# B&R Automation Studio project warcabot (part 2)

#### Types.typ
```iecst
TYPE
	CameraCommandType : 	STRUCT
		Enable : BOOL;
		AcquireImage : BOOL;
		SearchAcquisitionSettings : BOOL;
	END_STRUCT;
	BoardCalibrationType : 	STRUCT
		BottomRightY : DINT;
		BottomRightX : DINT;
		BottomLeftY : DINT;
		BottomLeftX : DINT;
		TopRightY : DINT;
		TopRightX : DINT;
		TopLeftY : DINT;
		TopLeftX : DINT;
		MarkersValid : BOOL;
		ReferenceMarker4Y : DINT;
		ReferenceMarker4X : DINT;
		ReferenceMarker3Y : DINT;
		ReferenceMarker3X : DINT;
		ReferenceBottomRightY : DINT;
		ReferenceBottomRightX : DINT;
		ReferenceBottomLeftY : DINT;
		ReferenceBottomLeftX : DINT;
		ReferenceTopRightY : DINT;
		ReferenceTopRightX : DINT;
		ReferenceTopLeftY : DINT;
		ReferenceTopLeftX : DINT;
	END_STRUCT;
	CameraParameterType : 	STRUCT
		FlashColor : USINT;
		FlashSegment : USINT;
		SetFocus : UINT;
		ExposureTime : UDINT;
		NumSearchMax : USINT;
		ScoreMin : USINT;
		GainLevel : USINT;
	END_STRUCT;
	CameraStatusType : 	STRUCT
		AcquisitionReady : BOOL;
		ProcessingActive : BOOL;
		ProcessingError : UINT;
		ReadFocus : UINT;
		ReadExposureTime : UDINT;
		ReadGainLevel : USINT;
	END_STRUCT;
	DetectedPieceType : 	STRUCT
		PositionX : DINT;
		PositionY : DINT;
		Valid : BOOL;
		Score : USINT;
		ModelNumber : USINT;
		Column : USINT;
		Row : USINT;
	END_STRUCT;
	CameraBoardType :ARRAY[1..8,1..8]OF USINT;
	CameraControlType : 	STRUCT
		Cmd : CameraCommandType;
		Parameters : CameraParameterType;
		Status : CameraStatusType;
		NumResults : USINT;
		Pieces : ARRAY[1..26]OF DetectedPieceType;
		Calibration : BoardCalibrationType;
		Board : CameraBoardType;
		BoardReady : BOOL;
		BlackCount : USINT;
		WhiteCount : USINT;
		BoardDataValid : BOOL;
	END_STRUCT;
END_TYPE
```

#### Variables.var
```iecst
VAR
	marker4X : DINT;
	marker3Y : DINT;
	marker3X : DINT;
	j : USINT;
	currentRightX : DINT;
	currentBoardWidth : DINT;
	currentLeftX : DINT;
	boardHeight : DINT;
	PreviousCameraAutoAdjust : BOOL;
	i : USINT;
	gCameraCtrl : CameraControlType;
	PreviousProcessingActive : BOOL;
	columnIndex : USINT;
	rowIndex : USINT;
	cellStepY : DINT;
	cellStepX : DINT;
	relativeY : DINT;
	relativeX : DINT;
	transformedY : LREAL;
	transformedX : LREAL;
	cornerRelativeY : LREAL;
	cornerRelativeX : LREAL;
	transformationDen : LREAL;
	transformationB : LREAL;
	transformationA : LREAL;
	currentVectorY : LREAL;
	currentVectorX : LREAL;
	referenceVectorY : LREAL;
	referenceVectorX : LREAL;
	marker4Found : BOOL;
	marker3Found : BOOL;
	marker4Y : DINT;
	PreviousAutoProcessingActive : BOOL;
END_VAR
```

#### Main.st
```iecst
PROGRAM _INIT

	gCameraCtrl.Cmd.Enable := TRUE;
	gCameraCtrl.Cmd.AcquireImage := FALSE;

	gCameraAutoAdjust := FALSE;
	PreviousCameraAutoAdjust := FALSE;

	gCameraExposureTime := 20884;
	gCameraGainLevel := 4;
	gCameraFocus := 53073;

	gCameraCtrl.Parameters.ExposureTime := gCameraExposureTime;
	gCameraCtrl.Parameters.SetFocus := gCameraFocus;
	gCameraCtrl.Parameters.GainLevel := gCameraGainLevel;
	gCameraCtrl.Parameters.FlashColor := 3;
	gCameraCtrl.Parameters.FlashSegment := 1;

	gCameraCtrl.Parameters.ScoreMin := 75;
	gCameraCtrl.Parameters.NumSearchMax := 26;

	gCameraCtrl.Calibration.ReferenceTopLeftX := 41009;
	gCameraCtrl.Calibration.ReferenceTopLeftY := 14517;
	gCameraCtrl.Calibration.ReferenceTopRightX := 120526;
	gCameraCtrl.Calibration.ReferenceTopRightY := 12412;

	gCameraCtrl.Calibration.ReferenceBottomLeftX := 41915;
	gCameraCtrl.Calibration.ReferenceBottomLeftY := 91572;

	gCameraCtrl.Calibration.ReferenceBottomRightX := 121154;
	gCameraCtrl.Calibration.ReferenceBottomRightY := 90368;

	gCameraCtrl.Calibration.ReferenceMarker3X := 41009;
	gCameraCtrl.Calibration.ReferenceMarker3Y := 14517;

	gCameraCtrl.Calibration.ReferenceMarker4X := 121154;
	gCameraCtrl.Calibration.ReferenceMarker4Y := 90368;

	gCameraCtrl.Calibration.MarkersValid := FALSE;

	gCameraCtrl.BoardReady := FALSE;
	gCameraCtrl.BoardDataValid := FALSE;
	gCameraCtrl.WhiteCount := 0;
	gCameraCtrl.BlackCount := 0;

	gCameraEnd := FALSE;
	PreviousProcessingActive := FALSE;

END_PROGRAM

PROGRAM _CYCLIC

	gCameraCtrl.Cmd.Enable := TRUE;

	(* Wyświetlanie rzeczywistych wartości kamery *)
	gCameraReadExposureTime :=
	gCameraCtrl.Status.ReadExposureTime;

	gCameraReadGainLevel :=
	gCameraCtrl.Status.ReadGainLevel;

	gCameraReadFocus :=
	gCameraCtrl.Status.ReadFocus;

	(* Po wyłączeniu ustawiania zapisz znalezione parametry *)
	IF PreviousCameraAutoAdjust AND NOT gCameraAutoAdjust THEN

		gCameraExposureTime :=
		gCameraCtrl.Status.ReadExposureTime;

		gCameraGainLevel :=
		gCameraCtrl.Status.ReadGainLevel;

		gCameraFocus :=
		gCameraCtrl.Status.ReadFocus;

	END_IF;

	(* Poza automatycznym ustawianiem wysyłaj zapisane nastawy *)
	IF NOT gCameraAutoAdjust THEN

		gCameraCtrl.Parameters.ExposureTime :=
		gCameraExposureTime;

		gCameraCtrl.Parameters.GainLevel :=
		gCameraGainLevel;

		gCameraCtrl.Parameters.SetFocus :=
		gCameraFocus;

	END_IF;

	PreviousCameraAutoAdjust := gCameraAutoAdjust;

	IF gCameraTrigger
		AND NOT gCameraAutoAdjust
		AND NOT gCameraEnd
		AND gCameraCtrl.Status.AcquisitionReady
		AND NOT gCameraCtrl.Status.ProcessingActive
		AND (gCameraCtrl.Status.ProcessingError = 0) THEN
		gCameraCtrl.Cmd.AcquireImage := TRUE;
	END_IF;

	gCameraBlackCount := gCameraCtrl.BlackCount;
	gCameraWhiteCount := gCameraCtrl.WhiteCount;
	gCameraNumResults := gCameraCtrl.NumResults;

	IF NOT gCameraTrigger THEN
		gCameraCtrl.Cmd.AcquireImage := FALSE;
		gCameraCtrl.BoardReady := FALSE;
		gCameraCtrl.BoardDataValid := FALSE;
		gCameraEnd := FALSE;
	END_IF;

	IF gCameraCtrl.Status.ProcessingActive THEN
		gCameraCtrl.Cmd.AcquireImage := FALSE;
	END_IF;

	IF gCameraTrigger
		AND PreviousProcessingActive
		AND NOT gCameraCtrl.Status.ProcessingActive THEN
		gCameraCtrl.Cmd.AcquireImage := FALSE;
		gCameraCtrl.BoardDataValid := TRUE;
		gCameraCtrl.WhiteCount := 0;
		gCameraCtrl.BlackCount := 0;
		marker3Found := FALSE;
		marker4Found := FALSE;
		cellStepY := 0;

		FOR rowIndex := 1 TO 8 DO
			FOR columnIndex := 1 TO 8 DO
				gCameraCtrl.Board[rowIndex, columnIndex] := 0;
			END_FOR;
		END_FOR;

		FOR i := 1 TO 26 DO
			IF gCameraCtrl.NumResults >= i THEN

				IF (gCameraCtrl.Pieces[i].ModelNumber = 3)
					AND (gCameraCtrl.Pieces[i].Score >= 30) THEN

					IF NOT marker3Found THEN

						marker3X := gCameraCtrl.Pieces[i].PositionX;
						marker3Y := gCameraCtrl.Pieces[i].PositionY;

						marker4X := gCameraCtrl.Pieces[i].PositionX;
						marker4Y := gCameraCtrl.Pieces[i].PositionY;

						marker3Found := TRUE;

					ELSE

						IF gCameraCtrl.Pieces[i].PositionX < marker3X THEN

							marker4X := marker3X;
							marker4Y := marker3Y;

							marker3X := gCameraCtrl.Pieces[i].PositionX;
							marker3Y := gCameraCtrl.Pieces[i].PositionY;

						ELSIF gCameraCtrl.Pieces[i].PositionX > marker4X THEN

							marker4X := gCameraCtrl.Pieces[i].PositionX;
							marker4Y := gCameraCtrl.Pieces[i].PositionY;

						END_IF;

						marker4Found := TRUE;

					END_IF;

				END_IF;

			END_IF;
		END_FOR;

		gCameraCtrl.Calibration.MarkersValid := marker3Found AND marker4Found;

		IF gCameraCtrl.Calibration.MarkersValid THEN
			referenceVectorX := DINT_TO_LREAL(gCameraCtrl.Calibration.ReferenceMarker4X- gCameraCtrl.Calibration.ReferenceMarker3X);

			referenceVectorY := DINT_TO_LREAL(gCameraCtrl.Calibration.ReferenceMarker4Y- gCameraCtrl.Calibration.ReferenceMarker3Y);

			currentVectorX := DINT_TO_LREAL(marker4X - marker3X);

			currentVectorY := DINT_TO_LREAL(marker4Y - marker3Y);

			transformationDen := (referenceVectorX * referenceVectorX) + (referenceVectorY * referenceVectorY);

			IF transformationDen > 0.0 THEN

				transformationA := ((currentVectorX * referenceVectorX) + (currentVectorY * referenceVectorY)) / transformationDen;

				transformationB := ((currentVectorY * referenceVectorX) - (currentVectorX * referenceVectorY)) / transformationDen;

				transformationDen := (transformationA * transformationA) + (transformationB * transformationB);

				IF transformationDen > 0.0 THEN

					boardHeight := ((gCameraCtrl.Calibration.ReferenceBottomLeftY - gCameraCtrl.Calibration.ReferenceTopLeftY) +
					(gCameraCtrl.Calibration.ReferenceBottomRightY - gCameraCtrl.Calibration.ReferenceTopRightY)) / 2;

					IF boardHeight > 0 THEN
						cellStepY := boardHeight / 7;
					ELSE
						gCameraCtrl.BoardDataValid := FALSE;
					END_IF;

				ELSE
					gCameraCtrl.BoardDataValid := FALSE;
				END_IF;

			ELSE
				gCameraCtrl.BoardDataValid := FALSE;
			END_IF;

		ELSE
			gCameraCtrl.BoardDataValid := FALSE;
		END_IF;

		FOR i := 1 TO 26 DO

			gCameraCtrl.Pieces[i].Valid :=
			(gCameraCtrl.NumResults >= i)
			AND
			(gCameraCtrl.Pieces[i].Score >= gCameraCtrl.Parameters.ScoreMin)
			AND
			((gCameraCtrl.Pieces[i].ModelNumber = 1)
			OR
			(gCameraCtrl.Pieces[i].ModelNumber = 2));

			IF gCameraCtrl.Pieces[i].Valid
				AND gCameraCtrl.Calibration.MarkersValid
				AND (cellStepY > 0)
				AND (transformationDen > 0.0) THEN

				cornerRelativeX := DINT_TO_LREAL(gCameraCtrl.Pieces[i].PositionX - marker3X);

				cornerRelativeY := DINT_TO_LREAL(gCameraCtrl.Pieces[i].PositionY - marker3Y);

				transformedX := DINT_TO_LREAL(gCameraCtrl.Calibration.ReferenceMarker3X) +
				((transformationA * cornerRelativeX) + (transformationB * cornerRelativeY)) / transformationDen;

				transformedY := DINT_TO_LREAL(gCameraCtrl.Calibration.ReferenceMarker3Y) +
				((-transformationB * cornerRelativeX) + (transformationA * cornerRelativeY)) / transformationDen;

				relativeY := LREAL_TO_DINT(transformedY) - gCameraCtrl.Calibration.ReferenceTopLeftY;

				IF relativeY < -(cellStepY / 2)
					OR relativeY > (boardHeight + (cellStepY / 2)) THEN

					gCameraCtrl.Pieces[i].Valid := FALSE;
					gCameraCtrl.BoardDataValid := FALSE;

				ELSE

					currentLeftX :=
					LREAL_TO_DINT(
						DINT_TO_LREAL(
					gCameraCtrl.Calibration.ReferenceTopLeftX
					)
					+
					(
					DINT_TO_LREAL(
					gCameraCtrl.Calibration.ReferenceBottomLeftX
					- gCameraCtrl.Calibration.ReferenceTopLeftX
					)
					*
					DINT_TO_LREAL(relativeY)
					)
					/
					DINT_TO_LREAL(boardHeight)
					);

					currentRightX :=
					LREAL_TO_DINT(
						DINT_TO_LREAL(
					gCameraCtrl.Calibration.ReferenceTopRightX
					)
					+
					(
					DINT_TO_LREAL(
					gCameraCtrl.Calibration.ReferenceBottomRightX
					- gCameraCtrl.Calibration.ReferenceTopRightX
					)
					*
					DINT_TO_LREAL(relativeY)
					)
					/
					DINT_TO_LREAL(boardHeight)
					);

					currentBoardWidth := currentRightX - currentLeftX;

					IF currentBoardWidth > 0 THEN
						cellStepX := currentBoardWidth / 7;
					ELSE
						cellStepX := 0;
						gCameraCtrl.Pieces[i].Valid := FALSE;
						gCameraCtrl.BoardDataValid := FALSE;
					END_IF;

					IF gCameraCtrl.Pieces[i].Valid
						AND (cellStepX > 0) THEN

						relativeX :=
						LREAL_TO_DINT(transformedX) - currentLeftX;

						IF relativeX < -(cellStepX / 2)
							OR relativeX > (currentBoardWidth + (cellStepX / 2)) THEN

							gCameraCtrl.Pieces[i].Valid := FALSE;
							gCameraCtrl.BoardDataValid := FALSE;

						ELSE

							gCameraCtrl.Pieces[i].Column := DINT_TO_USINT((relativeX + (cellStepX / 2)) / cellStepX) + 1;

							gCameraCtrl.Pieces[i].Row := 9 - (DINT_TO_USINT((relativeY + (cellStepY / 2)) / cellStepY) + 1);

							IF (gCameraCtrl.Pieces[i].Column = 0)
								OR (gCameraCtrl.Pieces[i].Column > 8)
								OR (gCameraCtrl.Pieces[i].Row = 0)
								OR (gCameraCtrl.Pieces[i].Row > 8) THEN

								gCameraCtrl.Pieces[i].Valid := FALSE;
								gCameraCtrl.BoardDataValid := FALSE;

							ELSIF gCameraCtrl.Board[
								gCameraCtrl.Pieces[i].Row,
								gCameraCtrl.Pieces[i].Column
								] <> 0 THEN

								gCameraCtrl.Pieces[i].Valid := FALSE;
								gCameraCtrl.BoardDataValid := FALSE;

							ELSE

								gCameraCtrl.Board[
								gCameraCtrl.Pieces[i].Row,
								gCameraCtrl.Pieces[i].Column
								] :=
								gCameraCtrl.Pieces[i].ModelNumber;

								IF gCameraCtrl.Pieces[i].ModelNumber = 1 THEN
									gCameraCtrl.WhiteCount :=
									gCameraCtrl.WhiteCount + 1;
								ELSE
									gCameraCtrl.BlackCount :=
									gCameraCtrl.BlackCount + 1;
								END_IF;

							END_IF;

						END_IF;

					END_IF;

				END_IF;

			ELSE
				gCameraCtrl.Pieces[i].Valid := FALSE;
			END_IF;

			IF NOT gCameraCtrl.Pieces[i].Valid THEN
				gCameraCtrl.Pieces[i].Row := 0;
				gCameraCtrl.Pieces[i].Column := 0;
			END_IF;

		END_FOR;

		FOR rowIndex := 1 TO 8 DO
			FOR columnIndex := 1 TO 8 DO
				gBoardCamera[rowIndex, columnIndex] :=
				gCameraCtrl.Board[rowIndex, columnIndex];
			END_FOR;
		END_FOR;

		gCameraCtrl.BoardReady :=
		gCameraCtrl.BoardDataValid
		AND (gCameraCtrl.Status.ProcessingError = 0);
		gCameraEnd := TRUE;
	END_IF;

	PreviousProcessingActive := gCameraCtrl.Status.ProcessingActive;

	IF gCameraTrigger
		AND (gCameraCtrl.Status.ProcessingError <> 0) THEN
		gCameraCtrl.Cmd.AcquireImage := FALSE;
		gCameraCtrl.BoardReady := FALSE;
		gCameraCtrl.BoardDataValid := FALSE;
		gCameraEnd := TRUE;
	END_IF;

END_PROGRAM

PROGRAM _EXIT

	gCameraCtrl.Cmd.AcquireImage := FALSE;
	gCameraCtrl.Cmd.Enable := FALSE;

	gCameraCtrl.BoardReady := FALSE;
	gCameraCtrl.BoardDataValid := FALSE;
	gCameraCtrl.Calibration.MarkersValid := FALSE;

	gCameraEnd := FALSE;
	PreviousProcessingActive := FALSE;
	PreviousCameraAutoAdjust := FALSE;
	gCameraAutoAdjust := FALSE;

END_PROGRAM
```

### Program Logical/Programs/SaveGame (IEC)

#### Main.st - Init, cyclic, exit code
```iecst
PROGRAM _INIT
	(* Włączenie Bloków Funkcyjnych MpRecipe *)
	MpRecipeXml_0(MpLink := ADR(MpLinkgRecipeSR), Enable := TRUE, DeviceName := ADR('SG'), FileName := ADR('Save'));
	MpRecipeRegPar_0(MpLink := ADR(MpLinkgRecipeSR), Enable := TRUE, PVName := ADR('SaveGame:Save'));

	(* Włączenie Bloków Funkcyjnych z UI *)
	MpRecipeUI_0(MpLink := ADR(MpLinkgRecipeSR), Enable := TRUE, DeviceName := ADR('SG'), UIConnect := ADR(UIConnect));
	UIConnect.Recipe.SortOrder := mpRECIPE_UI_SORT_DATE_DESCENDING;

END_PROGRAM

PROGRAM _CYCLIC
	(* Function Bloki *)
	MpRecipeXml_0();
	MpRecipeRegPar_0();
	MpRecipeUI_0();

	(* Czyszczenie komunikatów po otwrciu / zamknięciu okna *)
	IF NSDialogOpen THEN
		Saved := FALSE;
		InvSavFileName := FALSE;
		NSDialogOpen := FALSE;
	END_IF;

	CurrentFileName := UIConnect.Recipe.List.Names[UIConnect.Recipe.List.SelectedIndex];

	(* Sprawdzanie czy jest mniej plików niż max *)
	IndexOOR := UIConnect.Recipe.List.MaxSelection >= 19;
	NIndexOOR := UIConnect.Recipe.List.MaxSelection < 19;

	(* Zabezpieczenie przed ingerencją w Function Blok podczas jego pracy *)
	IF UIConnect.Status = mpRECIPE_UI_STATUS_IDLE THEN

		(* Jeśli przycisk New save kliknięty i jest mniej niż max plików
		sprawdź nazwę i możliwie stwórz nowy plik. Wyświetl komunikaty *)
		IF NewSave AND NOT IndexOOR THEN
			Saved := FALSE;
			InvSavFileName := FALSE;
			FB_ValidateFileName_0(sUserInput := SaveFileName);
			IF FB_ValidateFileName_0.bIsValid THEN
				Save.BoardActual := gBoardActual;
				Save.PlayerColor := gPlayerColor;
				Save.DifficultyLevel := gDifficultyLevel;
				Save.MoveHistory := gGameStats.MoveHistory;
				Save.MoveCount := gGameStats.MoveCount;

				UIConnect.New.FileName := FB_ValidateFileName_0.sValidName;
				UIConnect.New.Create := TRUE;
				SaveFileName := '';
				Saved := TRUE;
				NewSave := FALSE;
			ELSE
				InvSavFileName := TRUE;
				NewSave := FALSE;
			END_IF;

		END_IF;

		(* Ładowanie do zmiennej *)
		IF PreLoad THEN
			UIConnect.Recipe.Load := TRUE;
			PreLoad := FALSE;
		END_IF;

		(* Jeśli przycisk Load kliknięty przypisz zmienną z danymi do zmiennej globalnej *)
		IF Load THEN
			gBoardActual := Save.BoardActual;
			gPlayerColor := Save.PlayerColor;
			gDifficultyLevel := Save.DifficultyLevel;
			gGameStats.MoveHistory := Save.MoveHistory;
			gGameStats.MoveCount := Save.MoveCount;

			LoadingDone := TRUE;
			gStart := TRUE;
			gGameStats.Load := TRUE;
			Load := FALSE;
		END_IF;

		(* Jeśli przycisk Delete kliknięty usuń plik o wybranym indeksie *)
		IF DeleteSave THEN
			UIConnect.Recipe.Delete := TRUE;
			DeleteSave := FALSE;
		END_IF
	END_IF;

END_PROGRAM

PROGRAM _EXIT
	(* Wyłączenie Function Bloków *)
	MpRecipeXml_0(Enable := FALSE);
	MpRecipeRegPar_0(Enable := FALSE);
	MpRecipeUI_0(Enable := FALSE);

END_PROGRAM
```

#### Types.typ - Local data types
```iecst
TYPE
	Save_type : 	STRUCT
		BoardActual : ARRAY[1..8,1..8]OF USINT := [2,0,2,0,2,0,2,2(0),2,0,2,0,2,0,2(2),0,2,0,2,0,2,18(0),1,0,1,0,1,0,2(1),0,1,0,1,0,1,2(0),1,0,1,0,1,0,1];
		PlayerColor : BOOL := FALSE;
		MoveHistory : ARRAY[1..4]OF STRING[20];
		MoveCount : INT;
		DifficultyLevel : USINT := 0;
	END_STRUCT;
END_TYPE
```

#### Variables.var - Local variables
```iecst
VAR
	Load : BOOL := FALSE; (*Zmienna czy przycisk Save został kliknięty*)
	DeleteSave : BOOL := FALSE; (*Zmienna czy przycisk Delete został kliknięty*)
	MpRecipeXml_0 : MpRecipeXml;
	MpRecipeRegPar_0 : MpRecipeRegPar;
	MpRecipeUI_0 : MpRecipeUI; (*MpRecipeUI for UI Connection to the ice cream machine*)
	UIConnect : MpRecipeUIConnectType; (*UI Connection - interfejs do mprecipe*)
	Save : Save_type; (*Zmienna do której są zapisywane i z której są odczytywane dane*)
	SaveFileName : STRING[80]; (*Zmienna do przechowywania wpisanej nazwy pliku*)
	NewSave : BOOL := FALSE; (*Zmienna czy przycisk New save został kliknięty*)
	FB_ValidateFileName_0 : FB_ValidateFileName; (*Function Blok do sprawdzania czy nazwa pliku jest poprawna*)
	InvSavFileName : BOOL := FALSE; (*Zmienna do komunukacji o niepoprawnej nazwie*)
	Saved : BOOL := FALSE; (*Zmienna do komunikacji o pomyślnym zapisaniu pliku*)
	NSDialogOpen : BOOL := FALSE; (*Marker o otworzeniu okna New Save*)
	CurrentFileName : STRING[80]; (*Nazwa aktualnie wybranego pliku*)
	IndexOOR : BOOL; (*Marker o zapełnieniu listy (max 20 plików)*)
	NIndexOOR : BOOL; (*Negacja Markera IndexOOR*)
	LoadingDone : BOOL; (*Marker dla silnika gry*)
	PreLoad : BOOL; (*Zmienna czy przycisk Load (preLoead) został kliknięty*)
END_VAR
```

#### LocalFunctions.fun
```iecst
{REDUND_ERROR} FUNCTION_BLOCK FB_ValidateFileName (*Validating file name*) (*$GROUP=User,$CAT=User,$GROUPICON=User.png,$CATICON=User.png*)
	VAR_INPUT
		sUserInput : {REDUND_UNREPLICABLE} STRING[80]; (*Zmienna wejściowa ze sprawdzaną nazwą pliku*)
	END_VAR
	VAR_OUTPUT
		sValidName : STRING[80]; (*Zmienna wyjściowa z poprawną nazwą pliku*)
		bIsValid : BOOL; (*Zmienna informująca czy była możliwość dana poprawnej nazwy pliku na wyjściu*)
	END_VAR
	VAR
		i : UDINT; (*zmienna do iteracji po stringu*)
		tempChar : BYTE; (*Zmienna do przechowywania akutalnie iterownaje litery*)
	END_VAR
	VAR CONSTANT
		UNDERSCORE : BYTE := 95; (*ASCII value for '_'*)
	END_VAR
END_FUNCTION_BLOCK
```

#### FB_ValidateFileName.st
```iecst
(* TODO: Add your comment here *)
FUNCTION_BLOCK FB_ValidateFileName
(* Logic *)
	bIsValid := TRUE;
	sValidName := sUserInput;

	// 1. Check for empty input
	IF sUserInput = '' THEN
		bIsValid := FALSE;
	ELSE
		// 2. Sanitize string
		// We use LEN(sValidName) to get the current length of the string
		FOR i := 0 TO brsstrlen(ADR(sValidName)) - 1 DO
			// 1. READ: Copy current character from string into tempChar
			brsmemcpy(ADR(tempChar), ADR(sValidName) + i, 1);

			// 2. CHECK: Use tempChar for all comparisons
			IF tempChar = 32 THEN
				// WRITE: Copy underscore back into the string at position i
				brsmemcpy(ADR(sValidName) + i, ADR(UNDERSCORE), 1);

			ELSIF tempChar = 92 OR tempChar = 47 OR // \ and /
				tempChar = 58 OR tempChar = 42 OR // : and *
				tempChar = 63 OR tempChar = 34 OR // ? and "
				tempChar = 60 OR tempChar = 62 OR // < and >
				tempChar = 124 THEN               // |

				bIsValid := FALSE;
				EXIT;
			END_IF
		END_FOR
	END_IF
END_FUNCTION_BLOCK
```

### Program Logical/Programs/AlarmHistory (IEC)

#### Variables.var
```iecst
VAR
	AlarmTest : INT := 0; (*Testowa zmienna do testowania alarmów*)
	MpAlarmXHistory_0 : MpAlarmXHistory; (*Function blok MpAlarmXHistory*)
	AHExport : BOOL := FALSE; (*Zmienna czy przycisk export został kliknięty*)
	DirCreate_0 : DirCreate; (*Function Blok tworzący folder*)
	OpenExportDialog : BOOL := FALSE; (*Zmienna, która otwiera okienko z inf o exporcie*)
	AHClear : BOOL;
END_VAR
```

#### Main.st
```iecst
PROGRAM _INIT
	(* Włączenie Function Bloku MpAlarmXHistory *)
	MpAlarmXHistory_0(MpLink := ADR(MpLinkgAlarmXHistory), Enable := TRUE, DeviceName := ADR('AH'), FileName := ADR('Alarm_history'));

END_PROGRAM

PROGRAM _CYCLIC
	MpAlarmXHistory_0();

	(* Jeśli MpAlarmXHistory nic nie robi, a przycisk export kliknięty -> wyexportuj i otwórz okno dialogowe *)
	IF AHExport AND NOT MpAlarmXHistory_0.CommandBusy THEN
		MpAlarmXHistory_0.Export := TRUE;
		IF MpAlarmXHistory_0.CommandDone THEN
			MpAlarmXHistory_0.Export := FALSE;
			OpenExportDialog := TRUE;
			AHExport := FALSE;
		END_IF;
	END_IF;

	IF AHClear AND NOT MpAlarmXHistory_0.CommandBusy THEN
		MpAlarmXHistory_0.Clear := TRUE;
		IF MpAlarmXHistory_0.CommandDone THEN
			AHClear := FALSE;
		END_IF;
	END_IF;

END_PROGRAM

PROGRAM _EXIT
	(* Wyłacz MpAlarmXHistory *)
	MpAlarmXHistory_0(Enable := FALSE);

END_PROGRAM
```

### Program Logical/Programs/VisVariable (IEC)

#### Main.st
```iecst
PROGRAM _INIT
	gPickPiece;
	gEnableMove;
	gPickMove;
	gBoardActual;
	gGameRound;
	gEnablePiece;

END_PROGRAM

PROGRAM _CYCLIC
	(* Insert code here *)

END_PROGRAM

PROGRAM _EXIT
	(* Insert code here *)

END_PROGRAM
```

### Program Logical/Programs/GameStats (IEC)

#### Variables.var
```iecst
VAR
	WinOrLose : BOOL; (*True - wygrana, False - przegrana*)
	EndGame : BOOL; (*True - Koniec gry, False - gra wciaz trwa*)
	DeadWhitePiece : INT; (*Zbite biale pionki*)
	DeadBlackPiece : INT; (*Zbite czarne pionki*)
	MoveCount : INT; (*Ilosc ruchow*)
	i : USINT; (*zmienna do for*)
	j : USINT; (*zmienna do for*)
	whiteOnBoard : INT; (*ilosc bialych pionkow na planszy*)
	blackOnBoard : INT; (*ilosc czarnych pionkow na planszy*)
	gBoardLast : ARRAY[1..8,1..8] OF USINT; (*poprzedni stan planszy*)
	firstScan : BOOL := TRUE; (*pierwszy cykl - tylko zapamietaj plansze*)
	fromRow : USINT; (*wiersz startowy ruchu*)
	fromCol : USINT; (*kolumna startowa ruchu*)
	toRow : USINT; (*wiersz docelowy ruchu*)
	toCol : USINT; (*kolumna docelowa ruchu*)
	capCount : USINT; (*ilosc zbic w ruchu*)
	movedColor : USINT; (*1 - bialy, 2 - czarny*)
	cellColor : USINT; (*kolor pionka na polu*)
	pChar : REFERENCE TO USINT; (*wskaznik do budowy stringu*)
	LastMove : STRING[20]; (*ostatni wykryty ruch*)
	MoveHistory : ARRAY[1..4] OF STRING[20]; (*[1] najnowszy, [4] najstarszy*)
	MpAuditTrail_0 : MpAuditTrail;
	auditTmp : STRING[80];
	MessageVar : WSTRING[100];
	TypeVar : WSTRING[100];
	CommentVar : WSTRING[100];
	MpReportCore_0 : MpReportCore;
	sReport_Color     : STRING[20];
	sReport_Difficulty: STRING[30];
	sReport_Result    : STRING[20];
END_VAR
```

#### Main.st
```iecst
PROGRAM _INIT

	WinOrLose;
	EndGame;
	gPlayerColor;
	gDifficultyLevel;
	gStart;
	gBoardActual;
	j;
	i;
	whiteOnBoard;
	blackOnBoard;
	gEnablePiece;
	sReport_Color;
	sReport_Difficulty;
	sReport_Result;

	gBoardLast := gBoardActual;
	firstScan := TRUE;
	MoveHistory[1] := '';
	MoveHistory[2] := '';
	MoveHistory[3] := '';
	MoveHistory[4] := '';
	LastMove := '';
	MoveCount := 0;

	MpReportCore_0();
	MpReportCore_0.Enable := TRUE;
	MpReportCore_0.MpLink := ADR(gReport);
	MpReportCore_0.DeviceName := ADR('CF');
	MpReportCore_0.FileName := ADR('GameReport');
	MpReportCore_0.ReportID := ADR('MyReport');
	MpReportCore_0.Language := ADR('en');

END_PROGRAM

PROGRAM _CYCLIC

	MpReportCore_0();

	(* --- MAPOWANIE DANYCH NA TEKSTY --- *)

	(* Kolor *)
	IF gPlayerColor THEN
		sReport_Color := 'White';
	ELSE
		sReport_Color := 'Black';
	END_IF;

	(* Poziom trudności *)
	CASE gDifficultyLevel OF
		4: sReport_Difficulty := 'No stress';
		3: sReport_Difficulty := 'Easy going';
		0: sReport_Difficulty := 'Challenge';
		1: sReport_Difficulty := 'Blood, sweat & tears';
		2: sReport_Difficulty := 'Good luck ...';
		ELSE
			sReport_Difficulty := 'Unknown';
	END_CASE;

	(* Wynik *)
	IF WinOrLose THEN
		sReport_Result := 'Victory';
	ELSE
		sReport_Result := 'Defeat';
	END_IF;

	(* --- STEROWANIE GENEROWANIEM RAPORTU --- *)
	IF EndGame AND NOT MpReportCore_0.CommandBusy THEN
		MpReportCore_0.Generate := TRUE;
	ELSE
		MpReportCore_0.Generate := FALSE;
	END_IF;

	IF gStart THEN
		IF gGameStats.Load THEN
			MoveHistory := gGameStats.MoveHistory;
			MoveCount := gGameStats.MoveCount;
			gGameStats.Load := FALSE;
		END_IF;

		whiteOnBoard := 0;
		blackOnBoard := 0;

		FOR i := 1 TO 8 DO
			FOR j := 1 TO 8 DO
				CASE gBoardActual[i, j] OF
					1, 3:  whiteOnBoard := whiteOnBoard + 1;
					2, 4:  blackOnBoard := blackOnBoard + 1;
				END_CASE;
			END_FOR;
		END_FOR;

		DeadWhitePiece := 12 - whiteOnBoard;
		DeadBlackPiece := 12 - blackOnBoard;

		IF firstScan THEN
			gBoardLast := gBoardActual;
			firstScan := FALSE;
		ELSE
			fromRow := 0; fromCol := 0;
			toRow := 0;   toCol := 0;
			capCount := 0;
			movedColor := 0;

			FOR i := 1 TO 8 DO
				FOR j := 1 TO 8 DO
					IF gBoardLast[i, j] = 0 AND gBoardActual[i, j] <> 0 THEN
						toRow := i;
						toCol := j;
						IF gBoardActual[i, j] = 1 OR gBoardActual[i, j] = 3 THEN
							movedColor := 1;
						ELSE
							movedColor := 2;
						END_IF;
					END_IF;
				END_FOR;
			END_FOR;

			IF toRow <> 0 THEN
				FOR i := 1 TO 8 DO
					FOR j := 1 TO 8 DO
						IF gBoardLast[i, j] <> 0 AND gBoardActual[i, j] = 0 THEN
							IF gBoardLast[i, j] = 1 OR gBoardLast[i, j] = 3 THEN
								cellColor := 1;
							ELSE
								cellColor := 2;
							END_IF;

							IF cellColor = movedColor THEN
								fromRow := i;
								fromCol := j;
							ELSE
								capCount := capCount + 1;
							END_IF;
						END_IF;
					END_FOR;
				END_FOR;
			END_IF;

			IF toRow <> 0 AND fromRow <> 0 THEN

				gRobotMoveVar.StartPoint.x := fromCol;
				gRobotMoveVar.StartPoint.y := fromRow;
				gRobotMoveVar.EndPoint.x := toCol;
				gRobotMoveVar.EndPoint.y := toRow;
				gRobotMoveVar.RTRMove := TRUE;

				pChar ACCESS ADR(LastMove);
				pChar := 64 + fromCol;

				pChar ACCESS ADR(LastMove) + 1;
				pChar := 48 + fromRow;

				pChar ACCESS ADR(LastMove) + 2;
				IF capCount > 0 THEN
					pChar := 120;
					gRobotMoveVar.Capture := TRUE;
					gRobotMoveVar.DiscardPoint.x := (fromCol+toCol)/2;
					gRobotMoveVar.DiscardPoint.y := (fromRow+toRow)/2;
					gRobotMoveVar.DiscardColor := (movedColor) MOD 2 + 1;
				ELSE
					pChar := 45;
					gRobotMoveVar.Capture := FALSE;
				END_IF;

				pChar ACCESS ADR(LastMove) + 3;
				pChar := 64 + toCol;

				pChar ACCESS ADR(LastMove) + 4;
				pChar := 48 + toRow;

				pChar ACCESS ADR(LastMove) + 5;
				pChar := 0;

				MoveHistory[4] := MoveHistory[3];
				MoveHistory[3] := MoveHistory[2];
				MoveHistory[2] := MoveHistory[1];
				MoveHistory[1] := LastMove;

				MoveCount := MoveCount + 1;

				(* --- AUDIT: kto wykonal ruch i dokad --- *)
				IF movedColor = gPlayerColor THEN
					brsstrcpy(ADR(auditTmp), ADR('Gracz wykonal ruch: '));
				ELSE
					brsstrcpy(ADR(auditTmp), ADR('Robot wykonal ruch: '));
				END_IF;
				brsstrcat(ADR(auditTmp), ADR(LastMove));

				MessageVar := STRING_TO_WSTRING(auditTmp);
				TypeVar    := "GameMove";
				CommentVar := "";

				MpAuditCustomEvent(gAuditTrail, TypeVar, MessageVar, CommentVar);
				(* --- koniec AUDIT --- *)

				gGameStats.MoveHistory := MoveHistory;
				gGameStats.MoveCount := MoveCount;
			END_IF;

			gBoardLast := gBoardActual;
		END_IF;

	ELSE
		DeadWhitePiece := 0;
		DeadBlackPiece := 0;
		whiteOnBoard := 0;
		blackOnBoard := 0;
		MoveCount := 0;
		LastMove := '';
		MoveHistory[1] := '';
		MoveHistory[2] := '';
		MoveHistory[3] := '';
		MoveHistory[4] := '';
		firstScan := TRUE;
		gBoardLast := gBoardActual;
	END_IF

END_PROGRAM

PROGRAM _EXIT
    (* Insert code here *)

END_PROGRAM
```

### Program Logical/Programs/CheckVision (IEC)

#### Types.typ
```iecst
TYPE
	VisionEnum : 	STRUCT
		BoardConverted : ARRAY[1..8,1..8]OF USINT; (*Przekonwertowana tablica gdzie pokazywany jest tylko kolor, 1 - bialy, 2 - czarny, 0 -brak*)
		BoardVision : ARRAY[1..8,1..8]OF USINT; (*Tablica z kamery *)
		Step : StepVisionEnum; (*Kroki do case*)
		PhotoTake : BOOL; (*TRUE - kamera wykonala zdjecie*)
	END_STRUCT;
	StepVisionEnum :
		(
		CheckTable,
		ConvertTable
		);
END_TYPE
```

#### Variables.var
```iecst
VAR
	OUT : BOOL;
	j : USINT;
	i : USINT;
	Vision : VisionEnum;
	Match : BOOL;
END_VAR
```

#### Main.st
```iecst
PROGRAM _INIT
	gBoardActual;
	Vision;
	OUT := FALSE;

	Match;
	i;
	j;

	Vision.Step := ConvertTable;
	Vision.PhotoTake := FALSE;
END_PROGRAM

PROGRAM _CYCLIC

	CASE Vision.Step OF

		ConvertTable:
			FOR i := 1 TO 8 DO
				FOR j := 1 TO 8 DO
					CASE gBoardActual[i, j] OF
						1:  Vision.BoardConverted[i, j] := 1;
						2:  Vision.BoardConverted[i, j] := 2;
						3:  Vision.BoardConverted[i, j] := 1;
						4:  Vision.BoardConverted[i, j] := 2;
					END_CASE;
				END_FOR;
			END_FOR;

			IF Vision.PhotoTake THEN
				Vision.Step := CheckTable;
			END_IF;

		CheckTable:
			Match := TRUE;
			FOR i := 1 TO 8 DO
				FOR j := 1 TO 8 DO
					IF Vision.BoardConverted[i, j] <> Vision.BoardVision[i, j] THEN
						Match := FALSE;
					END_IF;
				END_FOR;
			END_FOR;

			IF Match THEN
				OUT := TRUE;
				Vision.Step := ConvertTable;
			ELSE
				Vision.Step := ConvertTable;
			END_IF;

	END_CASE

END_PROGRAM

PROGRAM _EXIT
	(* Insert code here *)

END_PROGRAM
```

### Program Logical/Programs/MainProgram (IEC)

#### Types.typ
```iecst
TYPE
	RobotMoveEnum :
		(
		IdleRM,
		MoveExecute,
		MoveBusy,
		DiscardExecute,
		DiscardBusy,
		HomeExecute,
		HomeBusy,
		EndRM
		);
	SetBoardInfoType : 	STRUCT
		Index : IndexPointType;
		Color : USINT; (*White = 1; Black = 2*)
	END_STRUCT;
	SetBoardEnum :
		(
		SetBoardCommandGen,
		SetBoardExecute,
		SetBoardBusy,
		SetBoardHomeExecute,
		SetBoardHomeBusy
		);
	CommandType : 	STRUCT
		EndPos : McPosType;
		StartPos : McPosType;
		EndIndex : IndexPointType;
		StartIndex : IndexPointType;
	END_STRUCT;
END_TYPE
```

#### Variables.var
```iecst
VAR
	ColorCount : ARRAY[1..2] OF USINT := [2(0)];
	MpAuditTrail_0 : MpAuditTrail;
	BoardGit : BOOL; (*Git ruch*)
	Match : BOOL;
	j : USINT;
	i : USINT;
	k : USINT;
	MoveStep : RobotMoveEnum := Idle;
	RobotMoveMarker : BOOL;
	MpReportCore_0 : MpReportCore;
	BuforLastPieceIndex : ARRAY[1..2] OF USINT;
	PiecesToDiscard : ARRAY[1..24] OF SetBoardInfoType;
	DiscardCount : USINT := 0;
	PiecesToDraw : ARRAY[1..24] OF SetBoardInfoType;
	DrawCount : USINT := 0;
	SimBoardValue : USINT := 0;
	CameraBoardValue : USINT := 0;
	DrawHandled : ARRAY[1..24] OF BOOL;
	DiscardHandled : ARRAY[1..24] OF BOOL;
	MatchFound : BOOL := FALSE;
	SetBoardStep : SetBoardEnum := SetBoardCommandGen;
	SetBoardTrigger : BOOL := FALSE;
	RRPCancel : BOOL := FALSE; (*Robot Reset Pos Cancel*)
	RRPConfirm : BOOL := FALSE; (*Robot Reset Pos Confirm*)
	CommandCount : USINT := 0;
	CommandList : ARRAY[1..48] OF CommandType;
	CommandDoneCount : USINT := 0;
	ReportLanguage : STRING[20] := 'en';
	RRPTrigger : BOOL;
END_VAR
VAR CONSTANT
	BOARD_SPACES : USINT := 8;
	CONVERT_BOARD : ARRAY[0..4] OF USINT := [0,1,2,1,2];
	BUFOR_POSITION : ARRAY[1..2,1..12] OF McPosType := [
	(X:=-61.8, Y:=68.9, Z:=-0.5),
	(X:=-28.1, Y:=69.0, Z:=-0.5),
	(X:=4.8, Y:=68.9, Z:=-0.5),
	(X:=-61.4, Y:=105.2, Z:=-0.7),
	(X:=-27.6, Y:=105.4, Z:=-0.8),
	(X:=4.3, Y:=105.2, Z:=-0.7),
	(X:=-61.5, Y:=141.4, Z:=-0.8),
	(X:=-28.4, Y:=141.5, Z:=-0.8),
	(X:=3.4, Y:=141.4, Z:=-0.8),
	(X:=-61.9, Y:=177.5, Z:=-0.9),
	(X:=-29.5, Y:=177.6, Z:=-0.9),
	(X:=2.2, Y:=177.5, Z:=-0.9),
	(X:=426.3, Y:=66.3, Z:=1.9),
	(X:=459.6, Y:=66.3, Z:=1.8),
	(X:=492.9, Y:=66.4, Z:=1.9),
	(X:=426.5, Y:=102.8, Z:=1.7),
	(X:=459.6, Y:=102.8, Z:=1.5),
	(X:=492.7, Y:=102.9, Z:=1.7),
	(X:=426.7, Y:=139.4, Z:=1.6),
	(X:=459.6, Y:=139.5, Z:=1.5),
	(X:=492.4, Y:=139.4, Z:=1.6),
	(X:=426.8, Y:=175.9, Z:=1.5),
	(X:=459.5, Y:=175.9, Z:=1.4),
	(X:=492.1, Y:=175.9, Z:=1.5)
	];
	COORD_POSITION : ARRAY[1..8,1..8] OF McPosType := [
	(X:=62.9, Y:=-29.7, Z:=2.4),
	(X:=107.2, Y:=-26.3, Z:=2.3),
	(X:=150.1, Y:=-26.9, Z:=2.5),
	(X:=193.0, Y:=-27.5, Z:=2.7),
	(X:=236.4, Y:=-28.7, Z:=2.4),
	(X:=278.7, Y:=-28.8, Z:=3.2),
	(X:=321.6, Y:=-29.4, Z:=3.4),
	(X:=363.6, Y:=-28.7, Z:=4.0),
	(X:=64.6, Y:=16.7, Z:=2.5),
	(X:=107.4, Y:=16.1, Z:=2.7),
	(X:=150.3, Y:=15.5, Z:=2.9),
	(X:=193.1, Y:=14.9, Z:=3.1),
	(X:=236.0, Y:=14.3, Z:=3.3),
	(X:=278.8, Y:=13.6, Z:=3.5),
	(X:=321.6, Y:=13.0, Z:=3.7),
	(X:=364.5, Y:=12.4, Z:=3.9),
	(X:=64.8, Y:=59.1, Z:=2.9),
	(X:=107.6, Y:=58.5, Z:=3.1),
	(X:=150.4, Y:=57.9, Z:=3.3),
	(X:=193.2, Y:=57.3, Z:=3.5),
	(X:=236.0, Y:=56.6, Z:=3.7),
	(X:=278.8, Y:=56.0, Z:=3.9),
	(X:=321.6, Y:=55.4, Z:=4.1),
	(X:=364.4, Y:=54.8, Z:=4.3),
	(X:=65.2, Y:=110.4, Z:=3.0),
	(X:=107.9, Y:=100.8, Z:=3.4),
	(X:=150.6, Y:=100.2, Z:=3.6),
	(X:=195.2, Y:=98.9, Z:=3.8),
	(X:=237.6, Y:=98.9, Z:=4.0),
	(X:=278.9, Y:=98.4, Z:=4.3),
	(X:=321.7, Y:=97.8, Z:=4.5),
	(X:=364.4, Y:=97.2, Z:=4.7),
	(X:=65.3, Y:=143.8, Z:=3.6),
	(X:=108.1, Y:=143.2, Z:=3.8),
	(X:=150.8, Y:=142.6, Z:=4.0),
	(X:=193.8, Y:=140.5, Z:=4.6),
	(X:=236.9, Y:=140.5, Z:=4.5),
	(X:=278.9, Y:=140.8, Z:=4.7),
	(X:=321.7, Y:=140.2, Z:=4.9),
	(X:=363.1, Y:=139.0, Z:=4.7),
	(X:=65.6, Y:=186.2, Z:=4.0),
	(X:=108.3, Y:=185.6, Z:=4.2),
	(X:=151.0, Y:=185.0, Z:=4.4),
	(X:=193.6, Y:=184.4, Z:=4.6),
	(X:=236.3, Y:=183.8, Z:=4.8),
	(X:=279.0, Y:=183.2, Z:=5.0),
	(X:=321.7, Y:=182.6, Z:=5.2),
	(X:=364.4, Y:=182.0, Z:=5.4),
	(X:=65.8, Y:=228.5, Z:=4.4),
	(X:=108.5, Y:=227.9, Z:=4.6),
	(X:=151.1, Y:=227.4, Z:=4.8),
	(X:=193.8, Y:=226.8, Z:=5.0),
	(X:=236.4, Y:=226.2, Z:=5.2),
	(X:=279.0, Y:=225.6, Z:=5.4),
	(X:=321.7, Y:=225.0, Z:=5.6),
	(X:=364.3, Y:=224.5, Z:=5.8),
	(X:=65.4, Y:=268.4, Z:=4.7),
	(X:=108.7, Y:=270.3, Z:=4.9),
	(X:=151.3, Y:=269.7, Z:=5.1),
	(X:=193.3, Y:=268.4, Z:=5.4),
	(X:=236.5, Y:=268.6, Z:=5.6),
	(X:=279.1, Y:=268.0, Z:=5.8),
	(X:=321.7, Y:=267.4, Z:=6.0),
	(X:=364.3, Y:=268.4, Z:=6.3)
	];
	DEFAULT_POSITION : McPosType := (X:=-139,Y:=359,Z:=350);
END_VAR
```

#### Main.st
```iecst
PROGRAM _INIT
	gStep := Idle;
	BoardGit := FALSE;

	MpAuditTrail_0.Enable := TRUE;
	MpAuditTrail_0.MpLink := ADR(gAuditTrail);
	MpAuditTrail_0.DeviceName := ADR('AUDIT');
	MpAuditTrail_0.FileName := ADR('AuditList');
	MpAuditTrail_0();
END_PROGRAM

PROGRAM _CYCLIC
	MpAuditTrail_0();

	gStop := NOT gStart;

	IF gESTOP = FALSE THEN
		gMotionInterface.Enable := FALSE;
	END_IF;

	IF gStart = FALSE THEN
		gStep := Idle;
		gRobotMoveVar.RTRMove := FALSE;
		MoveStep := IdleRM;
	END_IF;

	CASE gStep OF
		Idle:
			IF gStart THEN
				SetBoardTrigger := TRUE;
				gStep := ResetRobotPos;
				SetBoardStep := SetBoardBusy;
				gMotionInterface.Enable := TRUE;
				gMotionInterface.RequestManualMode := FALSE;
			END_IF;

		PhotoCheck:
			gCameraTrigger := TRUE;
			IF gCameraEnd THEN
				gCameraTrigger := FALSE;
				Match := TRUE;
				DrawCount := 0;
				DiscardCount := 0;
				ColorCount[1] := 0;
				ColorCount[2] := 0;

				FOR i := 1 TO BOARD_SPACES DO
					FOR j := 1 TO BOARD_SPACES DO
						(* Odwrócenie planszy do góry nogami, aby odczyt z kamery był zgodny z widokiem ze stania na wprost robota *)
						SimBoardValue := CONVERT_BOARD[gBoardActual[i, j]];
						CameraBoardValue := gBoardCamera[BOARD_SPACES + 1 - i, BOARD_SPACES + 1 - j];

						ColorCount[CameraBoardValue] := ColorCount[CameraBoardValue] + 1;

						IF SimBoardValue <> CameraBoardValue THEN
							Match := FALSE;

							IF SetBoardTrigger THEN
								IF CameraBoardValue = 0 THEN
									(* Inkrementujemy najpierw, aby zacząć od indeksu 1 *)
									DrawCount := DrawCount + 1;
									PiecesToDraw[DrawCount].Index.x := i;
									PiecesToDraw[DrawCount].Index.y := j;
									PiecesToDraw[DrawCount].Color := SimBoardValue;
								ELSIF SimBoardValue = 0 THEN
									(* Inkrementujemy najpierw, aby zacząć od indeksu 1 *)
									DiscardCount := DiscardCount + 1;
									PiecesToDiscard[DiscardCount].Index.x := i;
									PiecesToDiscard[DiscardCount].Index.y := j;
									PiecesToDiscard[DiscardCount].Color := CameraBoardValue;
								ELSE
									(* Zarówno w symulacji, jak i w kamerze jest pionek, ale RÓŻNYCH KOLORÓW -> ZAMIANA! *)
									(* 1. Najpierw usuwamy to, co fizycznie stoi na planszy (widzi to kamera) *)
									DiscardCount := DiscardCount + 1;
									PiecesToDiscard[DiscardCount].Index.x := i;
									PiecesToDiscard[DiscardCount].Index.y := j;
									PiecesToDiscard[DiscardCount].Color := CameraBoardValue;

									(* 2. Następnie stawiamy to, co powinno tam być zgodnie z symulacją *)
									DrawCount := DrawCount + 1;
									PiecesToDraw[DrawCount].Index.x := i;
									PiecesToDraw[DrawCount].Index.y := j;
									PiecesToDraw[DrawCount].Color := SimBoardValue;
								END_IF;
							END_IF;
						END_IF;
					END_FOR;
				END_FOR;

				IF Match THEN
					BoardGit := TRUE;
					gStep := GameMove;
				ELSE
					IF SetBoardTrigger THEN
						gStep := SetBoardPrep;
					ELSE
						gAlarm.InncorrectBoard := TRUE;
						gStep := ErrorState;
					END_IF;
				END_IF;
			END_IF;

		GameMove:
			(* GameMove -> wykonywany jest ruch warcabowy, gGameRound = TRUE -> ruch człowieka *)
			gPlayerMove := (gGameRound = TRUE);
			IF RobotMoveMarker AND gRobotMoveVar.RTRMove THEN
				gPlayerMove := FALSE;
				MoveStep := IdleRM;
				gStep := RobotMove;
				RobotMoveMarker := FALSE;
			END_IF;

		RobotMove:
			IF gESTOP THEN
				CASE MoveStep OF
					IdleRM:
						IF gRobotMoveVar.RTRMove THEN
							MoveStep := MoveExecute;
						END_IF;

					MoveExecute:
						IF gMotionInterface.Ready THEN
							gMotionInterface.Command := MOVE_START_END;
							gMotionInterface.StartPos := COORD_POSITION[gRobotMoveVar.StartPoint.y, gRobotMoveVar.StartPoint.x];
							gMotionInterface.EndPos := COORD_POSITION[gRobotMoveVar.EndPoint.y, gRobotMoveVar.EndPoint.x];
							gMotionInterface.Execute := TRUE;
							MoveStep := MoveBusy;
						END_IF;

					MoveBusy:
						IF gMotionInterface.Done THEN
							gMotionInterface.Execute := FALSE;
							IF gRobotMoveVar.Capture THEN
								MoveStep := DiscardExecute;
							ELSE
								MoveStep := HomeExecute;
							END_IF;
						END_IF;

					DiscardExecute:
						IF gMotionInterface.Ready THEN
							gMotionInterface.Command := MOVE_START_END;
							gMotionInterface.EndPos := BUFOR_POSITION[gRobotMoveVar.DiscardColor, 12 - ColorCount[gRobotMoveVar.DiscardColor] + 1];
							ColorCount[gRobotMoveVar.DiscardColor] := ColorCount[gRobotMoveVar.DiscardColor] - 1;
							gMotionInterface.StartPos := COORD_POSITION[gRobotMoveVar.DiscardPoint.y, gRobotMoveVar.DiscardPoint.x];
							gMotionInterface.Execute := TRUE;
							MoveStep := DiscardBusy;
						END_IF;

					DiscardBusy:
						IF gMotionInterface.Done THEN
							gMotionInterface.Execute := FALSE;
							MoveStep := HomeExecute;
						END_IF;

					HomeExecute:
						IF gMotionInterface.Ready THEN
							gMotionInterface.Command := MOVE_HOME;
							gMotionInterface.StartPos := DEFAULT_POSITION;
							gMotionInterface.EndPos := DEFAULT_POSITION;
							gMotionInterface.Execute := TRUE;
							MoveStep := HomeBusy;
						END_IF;

					HomeBusy:
						IF gMotionInterface.Done THEN
							gMotionInterface.Execute := FALSE;
							MoveStep := EndRM;
						END_IF;

					EndRM:
						MoveStep := IdleRM;
						gStep := PhotoCheck;
						gRobotMoveVar.RTRMove := FALSE;
				END_CASE;
			ELSE
				gStep := ResetRobotPos;
				SetBoardStep := SetBoardBusy;
				gRobotMoveVar.RTRMove := FALSE;
				MoveStep := IdleRM;
			END_IF;

		ErrorState:
			gMotionInterface.Enable := FALSE;
			IF gAlarm.InncorrectBoard = FALSE THEN
				gMotionInterface.Enable := TRUE;
				gStep := PhotoCheck;
			END_IF;

		ResetRobotPos:
			IF gESTOP THEN
				RRPTrigger := TRUE;
				IF RRPConfirm THEN
					CASE SetBoardStep OF
						SetBoardBusy:
							gMotionInterface.Enable := TRUE;
							SetBoardStep := SetBoardHomeExecute;

						SetBoardHomeExecute:
							IF gMotionInterface.Ready THEN
								gMotionInterface.Command := MOVE_HOME;
								gMotionInterface.StartPos := DEFAULT_POSITION;
								gMotionInterface.EndPos := DEFAULT_POSITION;
								gMotionInterface.Execute := TRUE;
								SetBoardStep := SetBoardHomeBusy;
							END_IF;

						SetBoardHomeBusy:
							IF gMotionInterface.Done THEN
								gMotionInterface.Execute := FALSE;
								RRPConfirm := FALSE;
								RRPTrigger := FALSE;
								SetBoardStep := SetBoardExecute;
								gStep := PhotoCheck;
							END_IF;
					END_CASE;
				ELSIF RRPCancel THEN
					gStart := FALSE;
					RRPCancel := FALSE;
					RRPTrigger := FALSE;
				END_IF;
			ELSE
				RRPConfirm := FALSE;
				RRPCancel := FALSE;
				RRPTrigger := FALSE;
			END_IF;

		SetBoardPrep:
			SetBoardTrigger := FALSE;

			(* Obliczanie aktualnego stanu bufora *)
			BuforLastPieceIndex[1] := 12 - ColorCount[1];
			BuforLastPieceIndex[2] := 12 - ColorCount[2];

			(* Zerowanie tablic flag *)
			FOR i := 1 TO 24 DO
				DrawHandled[i] := FALSE;
				DiscardHandled[i]:= FALSE;
			END_FOR;

			IF DrawCount > 0 OR DiscardCount > 0 THEN
				CommandCount := 0;

				(* KROK 1: Przesunięcia bezpośrednie z logiką antykolizyjną *)
				IF DiscardCount > 0 THEN
					FOR i := 1 TO DiscardCount DO
						IF NOT DiscardHandled[i] THEN
							MatchFound := FALSE;

							(* Szukamy wolnego miejsca o TAKIM SAMYM KOLORZE na planszy *)
							IF DrawCount > 0 THEN
								FOR j := 1 TO DrawCount DO
									IF NOT DrawHandled[j] AND (PiecesToDiscard[i].Color = PiecesToDraw[j].Color) THEN
										MatchFound := TRUE;

										(* --- LOGIKA ANTYKOLIZYJNA --- *)
										(* Sprawdzamy, czy na polu docelowym (PiecesToDraw[j]) fizycznie stoi jakiś inny błędny pionek *)
										FOR k := 1 TO DiscardCount DO
											IF (NOT DiscardHandled[k]) AND
												(PiecesToDiscard[k].Index.x = PiecesToDraw[j].Index.x) AND
												(PiecesToDiscard[k].Index.y = PiecesToDraw[j].Index.y) THEN

												(* ZNALEZIONO KOLIZJĘ! Najpierw odkładamy blokujący pionek do bufora *)
												CommandCount := CommandCount + 1;
												CommandList[CommandCount].StartPos := COORD_POSITION[PiecesToDiscard[k].Index.x, PiecesToDiscard[k].Index.y];

												IF BuforLastPieceIndex[PiecesToDiscard[k].Color] < 12 THEN
													BuforLastPieceIndex[PiecesToDiscard[k].Color] := BuforLastPieceIndex[PiecesToDiscard[k].Color] + 1;
												END_IF;

												CommandList[CommandCount].EndPos := BUFOR_POSITION[PiecesToDiscard[k].Color, BuforLastPieceIndex[PiecesToDiscard[k].Color]];

												(* Zaznaczamy, że ten blokujący pionek został już obsłużony *)
												DiscardHandled[k] := TRUE;
											END_IF;
										END_FOR;
										(* ----------------------------- *)

										(* Teraz pole docelowe jest NA PEWNO puste. Robimy ruch bezpośredni. *)
										CommandCount := CommandCount + 1;
										CommandList[CommandCount].StartPos := COORD_POSITION[PiecesToDiscard[i].Index.x, PiecesToDiscard[i].Index.y];
										CommandList[CommandCount].EndPos := COORD_POSITION[PiecesToDraw[j].Index.x, PiecesToDraw[j].Index.y];

										(* Oznaczamy jako obsłużone *)
										DiscardHandled[i] := TRUE;
										DrawHandled[j] := TRUE;
										EXIT; (* Przerywamy pętlę szukającą pary dla tego pionka *)
									END_IF;
								END_FOR;
							END_IF;

							(* Jeśli nie znaleźliśmy miejsca na planszy dla tego pionka (MatchFound = FALSE) -> zrzucamy do bufora *)
							IF NOT MatchFound THEN
								CommandCount := CommandCount + 1;
								CommandList[CommandCount].StartPos := COORD_POSITION[PiecesToDiscard[i].Index.x, PiecesToDiscard[i].Index.y];

								IF BuforLastPieceIndex[PiecesToDiscard[i].Color] < 12 THEN
									BuforLastPieceIndex[PiecesToDiscard[i].Color] := BuforLastPieceIndex[PiecesToDiscard[i].Color] + 1;
								END_IF;

								CommandList[CommandCount].EndPos := BUFOR_POSITION[PiecesToDiscard[i].Color, BuforLastPieceIndex[PiecesToDiscard[i].Color]];
								DiscardHandled[i] := TRUE;
							END_IF;
						END_IF;
					END_FOR;
				END_IF;

				(* KROK 2: Uzupełnianie brakujących miejsc (tych, które nie znalazły pary) z bufora *)
				IF DrawCount > 0 THEN
					FOR j := 1 TO DrawCount DO
						IF NOT DrawHandled[j] THEN
							CommandCount := CommandCount + 1;

							IF BuforLastPieceIndex[PiecesToDraw[j].Color] > 0 THEN
								CommandList[CommandCount].StartPos := BUFOR_POSITION[PiecesToDraw[j].Color, BuforLastPieceIndex[PiecesToDraw[j].Color]];
								BuforLastPieceIndex[PiecesToDraw[j].Color] := BuforLastPieceIndex[PiecesToDraw[j].Color] - 1;
							ELSE
								CommandList[CommandCount].StartPos := BUFOR_POSITION[PiecesToDraw[j].Color, 1];
							END_IF;

							CommandList[CommandCount].EndPos := COORD_POSITION[PiecesToDraw[j].Index.x, PiecesToDraw[j].Index.y];
							DrawHandled[j] := TRUE;
						END_IF;
					END_FOR;
				END_IF;

				CommandDoneCount := 0;
				gStep := SetBoard;
				SetBoardStep := SetBoardExecute;
			ELSE
				gStep := PhotoCheck;
			END_IF;

		SetBoard:
			IF gESTOP THEN
				CASE SetBoardStep OF
					SetBoardExecute:
						IF gMotionInterface.Ready THEN
							CommandDoneCount := CommandDoneCount + 1;
							gMotionInterface.Command := MOVE_START_END;
							gMotionInterface.StartPos := CommandList[CommandDoneCount].StartPos;
							gMotionInterface.EndPos := CommandList[CommandDoneCount].EndPos;
							gMotionInterface.Execute := TRUE;
							SetBoardStep := SetBoardBusy;
						END_IF;

					SetBoardBusy:
						IF gMotionInterface.Done THEN
							gMotionInterface.Execute := FALSE;

							IF CommandDoneCount < CommandCount THEN
								SetBoardStep := SetBoardExecute;
							ELSE
								SetBoardStep := SetBoardHomeExecute;
							END_IF;
						END_IF;

					SetBoardHomeExecute:
						IF gMotionInterface.Ready THEN
							gMotionInterface.Command := MOVE_HOME;
							gMotionInterface.StartPos := DEFAULT_POSITION;
							gMotionInterface.EndPos := DEFAULT_POSITION;
							gMotionInterface.Execute := TRUE;
							SetBoardStep := SetBoardHomeBusy;
						END_IF;

					SetBoardHomeBusy:
						IF gMotionInterface.Done THEN
							gMotionInterface.Execute := FALSE;
							SetBoardStep := SetBoardExecute;
							gStep := PhotoCheck;
						END_IF;
				END_CASE;
			ELSE
				SetBoardTrigger := FALSE;
				gStep := ResetRobotPos;
				SetBoardStep := SetBoardBusy;
			END_IF;
	END_CASE;
END_PROGRAM

PROGRAM _EXIT
	(* Miejsce na kod wywoływany przy zatrzymaniu zadania *)
END_PROGRAM
```

### Program Logical/Programs/FolderMng (IEC)

#### Variables.var
```iecst
VAR
	step : UINT := 10;
	strPath : STRING;

	(* FUBs *)
	fbDirCreate : DirCreate;
	fbDirInfo : DirInfo;
END_VAR
```

#### Main.st
```iecst
PROGRAM _INIT
	step := 10;
END_PROGRAM

PROGRAM _CYCLIC
	CASE step OF

		10: (* CHECK: 'Programs' folder exists AND has exactly 2 files *)
			strPath := 'Programs';
			fbDirInfo.enable := TRUE;
			fbDirInfo.pDevice := ADR('USER');
			fbDirInfo.pPath := ADR(strPath);
			fbDirInfo();

			IF fbDirInfo.status = 0 THEN
				IF fbDirInfo.filenum <> 3 THEN
					gAlarm.MissingSTMotionProgram := TRUE;
				ELSE
					gAlarm.MissingSTMotionProgram := FALSE;
				END_IF;
				step := 20;

			ELSIF fbDirInfo.status = 20723 THEN
				step := 100;

			ELSIF fbDirInfo.status <> 65535 THEN
				gAlarm.FolderError := TRUE;
				step := 20;
			END_IF;

		20: (* CHECK: 'SavedGames' folder exists *)
			strPath := 'SavedGames';
			fbDirInfo.enable := TRUE;
			fbDirInfo.pDevice := ADR('USER');
			fbDirInfo.pPath := ADR(strPath);
			fbDirInfo();

			IF fbDirInfo.status = 0 THEN
				step := 30;

			ELSIF fbDirInfo.status = 20723 THEN
				step := 110;

			ELSIF fbDirInfo.status <> 65535 THEN
				gAlarm.FolderError := TRUE;
				step := 30;
			END_IF;

		30: (* CHECK: 'AlarmHistory' folder exists *)
			strPath := 'AlarmHistory';
			fbDirInfo.enable := TRUE;
			fbDirInfo.pDevice := ADR('USER');
			fbDirInfo.pPath := ADR(strPath);
			fbDirInfo();

			IF fbDirInfo.status = 0 THEN
				step := 40;

			ELSIF fbDirInfo.status = 20723 THEN
				step := 120;

			ELSIF fbDirInfo.status <> 65535 THEN
				gAlarm.FolderError := TRUE;
				step := 40;
			END_IF;

		40: (* CHECK: 'Report' folder exists *)
			strPath := 'Report';
			fbDirInfo.enable := TRUE;
			fbDirInfo.pDevice := ADR('USER');
			fbDirInfo.pPath := ADR(strPath);
			fbDirInfo();

			IF fbDirInfo.status = 0 THEN
				step := 50;

			ELSIF fbDirInfo.status = 20723 THEN
				step := 130;

			ELSIF fbDirInfo.status <> 65535 THEN
				gAlarm.FolderError := TRUE;
				step := 50;
			END_IF;

		50: (* CHECK: 'Audit' folder exists *)
			strPath := 'Audit';
			fbDirInfo.enable := TRUE;
			fbDirInfo.pDevice := ADR('USER');
			fbDirInfo.pPath := ADR(strPath);
			fbDirInfo();

			IF fbDirInfo.status = 0 THEN
				step := 60;

			ELSIF fbDirInfo.status = 20723 THEN
				step := 140;

			ELSIF fbDirInfo.status <> 65535 THEN
				gAlarm.FolderError := TRUE;
				step := 60;
			END_IF;

		60: (* Loop reset *)
			step := 10;

			(* ===================== *)
			(* CREATION SEQUENCE     *)
			(* ===================== *)

		100: (* Create Programs *)
			strPath := 'Programs';
			fbDirCreate.enable := TRUE;
			fbDirCreate.pDevice := ADR('USER');
			fbDirCreate.pName := ADR(strPath);
			fbDirCreate();

			IF fbDirCreate.status = 0 THEN
				step := 10;
			ELSIF fbDirCreate.status <> 65535 THEN
				step := 999;
			END_IF;

		110: (* Create SavedGames *)
			strPath := 'SavedGames';
			fbDirCreate.enable := TRUE;
			fbDirCreate.pDevice := ADR('USER');
			fbDirCreate.pName := ADR(strPath);
			fbDirCreate();

			IF fbDirCreate.status = 0 THEN
				step := 20;
			ELSIF fbDirCreate.status <> 65535 THEN
				step := 999;
			END_IF;

		120: (* Create AlarmHistory *)
			strPath := 'AlarmHistory';
			fbDirCreate.enable := TRUE;
			fbDirCreate.pDevice := ADR('USER');
			fbDirCreate.pName := ADR(strPath);
			fbDirCreate();

			IF fbDirCreate.status = 0 THEN
				step := 30;
			ELSIF fbDirCreate.status <> 65535 THEN
				step := 999;
			END_IF;

		130: (* Create Report *)
			strPath := 'Report';
			fbDirCreate.enable := TRUE;
			fbDirCreate.pDevice := ADR('USER');
			fbDirCreate.pName := ADR(strPath);
			fbDirCreate();

			IF fbDirCreate.status = 0 THEN
				step := 40;
			ELSIF fbDirCreate.status <> 65535 THEN
				step := 999;
			END_IF;

		140: (* Create Audit *)
			strPath := 'Audit';
			fbDirCreate.enable := TRUE;
			fbDirCreate.pDevice := ADR('USER');
			fbDirCreate.pName := ADR(strPath);
			fbDirCreate();

			IF fbDirCreate.status = 0 THEN
				step := 50;
			ELSIF fbDirCreate.status <> 65535 THEN
				step := 999;
			END_IF;

		999: (* Error *)
			gAlarm.FolderError := TRUE;
			step := 10;

	END_CASE;
END_PROGRAM

PROGRAM _EXIT
  (* Insert code here *)

END_PROGRAM
```

### Program Logical/Programs/CheckLegal (IEC)

#### Main.st - Init, cyclic, exit code
```iecst
PROGRAM _INIT
	MoveLegal := FALSE;
	PlayerColor := WHITE_COLOR;
	gTest := FALSE;
END_PROGRAM

PROGRAM _CYCLIC
	IF gTest THEN

		MoveLegal := CanPlayerCapture(
		PlayerColor := PlayerColor,
		Board := gBoardBoard);

		gTest := FALSE;

	END_IF;
END_PROGRAM

PROGRAM _EXIT
	(* Insert code here *)

END_PROGRAM
```

#### Variables.var - Local variables
```iecst
VAR
	MoveLegal : BOOL;
	Piece : PieceTypeEnum;
	PlayerColor : PlayerColorEnum;
END_VAR
```

#### LocalFunctions.fun
```iecst
{REDUND_ERROR} FUNCTION CheckMove : BOOL (*TODO: Add your comment here*) (*$GROUP=User,$CAT=User,$GROUPICON=User.png,$CATICON=User.png*)
	VAR_INPUT
		FromRow : INT;
		FromColumn : INT;
		ToRow : INT;
		ToColumn : INT;
		Piece : PieceTypeEnum;
		Board : ARRAY[1..8,1..8] OF PieceTypeEnum;
	END_VAR
	VAR
		RowDiff : INT;
		ColDiff : INT;
	END_VAR
END_FUNCTION

{REDUND_ERROR} FUNCTION CheckRegularCapture : BOOL (*TODO: Add your comment here*) (*$GROUP=User,$CAT=User,$GROUPICON=User.png,$CATICON=User.png*)
	VAR_INPUT
		FromRow : INT;
		FromColumn : INT;
		ToRow : INT;
		ToColumn : INT;
		Piece : PieceTypeEnum;
		Board : ARRAY[1..8,1..8] OF PieceTypeEnum;
	END_VAR
	VAR
		MiddlePiece : PieceTypeEnum;
		RowDiff : INT;
		ColDiff : INT;
		MiddleRow : INT;
		MiddleColumn : INT;
	END_VAR
END_FUNCTION

{REDUND_ERROR} FUNCTION CanPlayerCapture : BOOL (*TODO: Add your comment here*) (*$GROUP=User,$CAT=User,$GROUPICON=User.png,$CATICON=User.png*)
	VAR_INPUT
		PlayerColor : PlayerColorEnum;
		Board : ARRAY[1..8,1..8] OF PieceTypeEnum;
	END_VAR
	VAR
		Row : INT;
		Column : INT;
		Piece : PieceTypeEnum;
		WHITE_PLAYER : BOOL;
		BLACK_PLAYER : BOOL;
	END_VAR
END_FUNCTION
```

#### CheckMove.st
```iecst
(* TODO: Add your comment here *)
FUNCTION CheckMove

	CheckMove := FALSE;

	(* Sprawdzenie zakresu planszy *)
	IF (FromRow < 1) OR (FromRow > 8) OR
		(FromColumn < 1) OR (FromColumn > 8) OR
		(ToRow < 1) OR (ToRow > 8) OR
		(ToColumn < 1) OR (ToColumn > 8) THEN
		RETURN;
	END_IF;

	(* Pole początkowe nie może być puste *)
	IF Piece = EMPTY THEN
		RETURN;
	END_IF;

	(* Pole docelowe musi być puste *)
	IF Board[ToRow, ToColumn] <> EMPTY THEN
		RETURN;
	END_IF;

	RowDiff := ToRow - FromRow;
	ColDiff := ToColumn - FromColumn;

	CASE Piece OF

		WHITE:

			IF (RowDiff = 1) AND
				((ColDiff = 1) OR (ColDiff = -1)) THEN
				CheckMove := TRUE;
			END_IF;

		BLACK:

			IF (RowDiff = -1) AND
				((ColDiff = 1) OR (ColDiff = -1)) THEN
				CheckMove := TRUE;
			END_IF;

	END_CASE;

END_FUNCTION
```

#### CheckRegularCapture.st
```iecst
(* TODO: Add your comment here *)
FUNCTION CheckRegularCapture

	CheckRegularCapture := FALSE;

	(* Sprawdzenie zakresu planszy *)
	IF (FromRow < 1) OR (FromRow > 8) OR
		(FromColumn < 1) OR (FromColumn > 8) OR
		(ToRow < 1) OR (ToRow > 8) OR
		(ToColumn < 1) OR (ToColumn > 8) THEN
		RETURN;
	END_IF;

	(* Pole początkowe nie może być puste *)
	IF Piece = EMPTY THEN
		RETURN;
	END_IF;

	(* Pole docelowe musi być puste *)
	IF Board[ToRow, ToColumn] <> EMPTY THEN
		RETURN;
	END_IF;

	RowDiff := ToRow - FromRow;
	ColDiff := ToColumn - FromColumn;

	CASE Piece OF

		WHITE:

			IF (RowDiff = 2) AND
				((ColDiff = 2) OR (ColDiff = -2)) THEN

				MiddleRow := FromRow + 1;
				MiddleColumn := FromColumn + (ColDiff / 2);

				MiddlePiece := Board[MiddleRow, MiddleColumn];

				IF (MiddlePiece = BLACK) OR
					(MiddlePiece = BLACK_KING) THEN
					CheckRegularCapture := TRUE;
				END_IF;

			END_IF;

		BLACK:

			IF (RowDiff = -2) AND
				((ColDiff = 2) OR (ColDiff = -2)) THEN

				MiddleRow := FromRow - 1;
				MiddleColumn := FromColumn + (ColDiff / 2);

				MiddlePiece := Board[MiddleRow, MiddleColumn];

				IF (MiddlePiece = WHITE) OR
					(MiddlePiece = WHITE_KING) THEN
					CheckRegularCapture := TRUE;
				END_IF;

			END_IF;

			WHITE_KING,
		BLACK_KING:

			IF ((RowDiff = 2) OR (RowDiff = -2)) AND
				((ColDiff = 2) OR (ColDiff = -2)) THEN

				MiddleRow := (FromRow + ToRow) / 2;
				MiddleColumn := (FromColumn + ToColumn) / 2;

				MiddlePiece := Board[MiddleRow, MiddleColumn];

				IF ((Piece = WHITE_KING) AND
					((MiddlePiece = BLACK) OR (MiddlePiece = BLACK_KING)))
					OR
					((Piece = BLACK_KING) AND
					((MiddlePiece = WHITE) OR (MiddlePiece = WHITE_KING))) THEN

					CheckRegularCapture := TRUE;

				END_IF;

			END_IF;

	END_CASE;

END_FUNCTION
```

### Program Logical/Programs/ManualCtrl

#### Variables.var
```iecst
VAR
	gRobotJog : MpGroupJog;
	gRobotJogPar : MpGroupJogParType;
END_VAR
```

#### Main.st
```iecst
PROGRAM _INIT
	(* Insert code here *)

END_PROGRAM

PROGRAM _CYCLIC

END_PROGRAM

PROGRAM _EXIT
	(* Insert code here *)

END_PROGRAM
```

### Library Logical/Programs/MovePiece

#### LocalFunctions.fun
```iecst
{REDUND_ERROR} {REDUND_UNREPLICABLE} FUNCTION_BLOCK FB_MovePiece (*TODO: Add your comment here*) (*$GROUP=User,$CAT=User,$GROUPICON=User.png,$CATICON=User.png*)
	VAR_INPUT
		Execute : {REDUND_UNREPLICABLE} BOOL;
	END_VAR
	VAR_OUTPUT
		Done : {REDUND_UNREPLICABLE} BOOL;
		Error : {REDUND_UNREPLICABLE} BOOL;
		ErrorID : {REDUND_UNREPLICABLE} INT;
	END_VAR
	VAR
		Piece : {REDUND_UNREPLICABLE} PieceTypeEnum;
		OldPosition : {REDUND_UNREPLICABLE} PositionStruct;
		NewPosition : {REDUND_UNREPLICABLE} PositionStruct;
		Piece1 : BOOL;
		gBoardBoard : BOOL;
		gCurrentMove : structType;
		gBoard : BOOL;
	END_VAR
END_FUNCTION_BLOCK
```

#### FB_MovePiece.st
```iecst
(* TODO: Add your comment here *)
FUNCTION_BLOCK FB_MovePiece
	Piece := gBoardBoard[gCurrentMove.FromRow, gCurrentMove.FromColumn];
	gBoardBoard[gCurrentMove.ToRow, gCurrentMove.ToColumn] := Piece;
	gBoard[gCurrentMove.FromRow, gCurrentMove.FromColumn] := EMPTY;
	gMoveCounter := gMoveCounter + 1;
END_FUNCTION_BLOCK
```

### Program Logical/Programs/PieceMovementProgram (IEC)

#### Test.st - Init, cyclic, exit code
```iecst
PROGRAM _INIT

	bInitGame := FALSE;
	bInitBoard := FALSE;
	bMovePiece := FALSE;
	bTest := FALSE;

END_PROGRAM

PROGRAM _CYCLIC

	instInitGame(
		Execute := bInitGame,
		MovesWithoutCapture := gMovesWithoutCapture,
		PlayerColor := gPlayerColor,
		Winner := gWinner,
		GameState := gGameState
	);

	instInitBoard(
		Execute := bInitBoard,
		BoardBoard := gBoardBoard,
		GameState := gGameState
	);

	instMovePiece(
		Execute := bMovePiece,
		FromRow := gCurrentMove.FROM_ROW,
		FromColumn := gCurrentMove.FROM_COLUMN,
		ToRow := gCurrentMove.TO_ROW,
		ToColumn := gCurrentMove.TO_COLUMN,
		Board := gBoardBoard
	);

	IF instMovePiece.Done THEN
		bMovePiece := FALSE; (* Wyłączamy trigger, aby nie wykonać ruchu ponownie w następnym cyklu *)
	END_IF;

	instPromotePiece(
		Execute := TRUE,
		Row := gCurrentMove.TO_ROW,
		Column := gCurrentMove.TO_COLUMN,
		Board := gBoardBoard
	);

	IF bTest THEN

		stCurrentPiece := gBoardBoard[gCurrentMove.TO_ROW, gCurrentMove.TO_COLUMN];

		bCanCaptureAgain := CanPieceCaptureAgain(
		Row := gCurrentMove.TO_ROW,      (* Nowy wiersz po ruchu *)
		Column := gCurrentMove.TO_COLUMN,   (* Nowa kolumna po ruchu *)
		Piece := stCurrentPiece,
		Board := gBoardBoard
		);

	END_IF;

END_PROGRAM

PROGRAM _EXIT

END_PROGRAM
```

#### Variables.var - Local variables
```iecst
VAR
	Piece : PieceTypeEnum;
	instMovePiece : FB_MovePiece;
	MoveLegal : BOOL;
END_VAR
```

#### LocalFunctions.fun
```iecst
{REDUND_ERROR} FUNCTION CanPlayerCapture : BOOL (*TODO: Add your comment here*) (*$GROUP=User,$CAT=User,$GROUPICON=User.png,$CATICON=User.png*)
	VAR_INPUT
		PlayerColor : PlayerColorEnum;
		Board : ARRAY[1..8,1..8] OF PieceTypeEnum;
	END_VAR
	VAR
		Row : INT;
		Column : INT;
		Piece : PieceTypeEnum;
		WHITE_PLAYER : BOOL;
		BLACK_PLAYER : BOOL;
	END_VAR
END_FUNCTION

{REDUND_ERROR} FUNCTION CheckMove : BOOL (*TODO: Add your comment here*) (*$GROUP=User,$CAT=User,$GROUPICON=User.png,$CATICON=User.png*)
	VAR_INPUT
		FromRow : INT;
		FromColumn : INT;
		ToRow : INT;
		ToColumn : INT;
		Piece : PieceTypeEnum;
		Board : ARRAY[1..8,1..8] OF PieceTypeEnum;
	END_VAR
	VAR
		RowDiff : INT;
		ColDiff : INT;
	END_VAR
END_FUNCTION

{REDUND_ERROR} FUNCTION CheckRegularCapture : BOOL (*TODO: Add your comment here*) (*$GROUP=User,$CAT=User,$GROUPICON=User.png,$CATICON=User.png*)
	VAR_INPUT
		FromRow : INT;
		FromColumn : INT;
		ToRow : INT;
		ToColumn : INT;
		Piece : PieceTypeEnum;
		Board : ARRAY[1..8,1..8] OF PieceTypeEnum;
	END_VAR
	VAR
		MiddlePiece : PieceTypeEnum;
		RowDiff : INT;
		ColDiff : INT;
		MiddleRow : INT;
		MiddleColumn : INT;
	END_VAR
END_FUNCTION

{REDUND_ERROR} {REDUND_UNREPLICABLE} FUNCTION_BLOCK FB_InitGame (*TODO: Add your comment here*) (*$GROUP=User,$CAT=User,$GROUPICON=User.png,$CATICON=User.png*)
	VAR_INPUT
		Execute : {REDUND_UNREPLICABLE} BOOL;
	END_VAR
	VAR_OUTPUT
		Done : {REDUND_UNREPLICABLE} BOOL;
	END_VAR
	VAR_IN_OUT
		MovesWithoutCapture : INT;
		PlayerColor : PlayerColorEnum;
		Winner : WinnerEnum;
		GameState : GameStateEnum;
	END_VAR
END_FUNCTION_BLOCK

FUNCTION_BLOCK FB_MovePiece
	VAR_INPUT
		Execute : BOOL;
		FromRow : INT;
		FromColumn : INT;
		ToRow : INT;
		ToColumn : INT;
		Piece : PieceTypeEnum; (* Dodaj to tutaj! *)
	END_VAR
	VAR_OUTPUT
		Done : BOOL; (* Teraz Done jest poprawnym wyjściem *)
	END_VAR
	VAR_IN_OUT
		Board : ARRAY[1..8,1..8] OF PieceTypeEnum;
	END_VAR
END_FUNCTION_BLOCK

{REDUND_ERROR} FUNCTION_BLOCK FB_InitBoard (*TODO: Add your comment here*) (*$GROUP=User,$CAT=User,$GROUPICON=User.png,$CATICON=User.png*)
	VAR_INPUT
		Execute : {REDUND_UNREPLICABLE} BOOL;
	END_VAR
	VAR_OUTPUT
		Done : BOOL;
	END_VAR
	VAR_IN_OUT
		BoardBoard : ARRAY[1..8,1..8] OF PieceTypeEnum;
		GameState : GameStateEnum;
	END_VAR
	VAR
		Row : INT;
		Column : INT;
	END_VAR
END_FUNCTION_BLOCK

{REDUND_ERROR} FUNCTION CanPieceCaptureAgain : BOOL (*TODO: Add your comment here*) (*$GROUP=User,$CAT=User,$GROUPICON=User.png,$CATICON=User.png*)
	VAR_INPUT
		Row : INT;
		Column : INT;
		Piece : PieceTypeEnum;
		Board : ARRAY[1..8,1..8] OF PieceTypeEnum;
	END_VAR
END_FUNCTION

{REDUND_ERROR} FUNCTION_BLOCK FB_PromotePiece (*TODO: Add your comment here*) (*$GROUP=User,$CAT=User,$GROUPICON=User.png,$CATICON=User.png*)
	VAR_INPUT
		Execute : BOOL;
		Row : INT;
		Column : INT;
	END_VAR

	VAR_OUTPUT
		Done : BOOL;
	END_VAR

	VAR_IN_OUT
		Board : ARRAY[1..8,1..8] OF PieceTypeEnum;
	END_VAR
END_FUNCTION_BLOCK
```

#### FB_MovePiece.st
```iecst
FUNCTION_BLOCK FB_MovePiece

	IF Execute THEN
		(* Zastąp gBoardBoard przez Board *)
		Piece := Board[FromRow, FromColumn];
		Board[ToRow, ToColumn] := Piece;
		Board[FromRow, FromColumn] := EMPTY;
		Done := TRUE;
	END_IF;

END_FUNCTION_BLOCK
```

#### CheckMove.st
```iecst
(* TODO: Add your comment here *)
FUNCTION CheckMove

	CheckMove := FALSE;

	(* Sprawdzenie zakresu planszy *)
	IF (FromRow < 1) OR (FromRow > 8) OR
		(FromColumn < 1) OR (FromColumn > 8) OR
		(ToRow < 1) OR (ToRow > 8) OR
		(ToColumn < 1) OR (ToColumn > 8) THEN
		RETURN;
	END_IF;

	(* Pole początkowe nie może być puste *)
	IF Piece = EMPTY THEN
		RETURN;
	END_IF;

	(* Pole docelowe musi być puste *)
	IF Board[ToRow, ToColumn] <> EMPTY THEN
		RETURN;
	END_IF;

	RowDiff := ToRow - FromRow;
	ColDiff := ToColumn - FromColumn;

	CASE Piece OF

		WHITE:

			IF (RowDiff = 1) AND
				((ColDiff = 1) OR (ColDiff = -1)) THEN
				CheckMove := TRUE;
			END_IF;

		BLACK:

			IF (RowDiff = -1) AND
				((ColDiff = 1) OR (ColDiff = -1)) THEN
				CheckMove := TRUE;
			END_IF;

		WHITE_KING,
		BLACK_KING:

			IF ((RowDiff = 1) OR (RowDiff = -1)) AND
				((ColDiff = 1) OR (ColDiff = -1)) THEN
				CheckMove := TRUE;
			END_IF;

	END_CASE;

END_FUNCTION
```

#### CanPlayerCapture.st
```iecst
(* TODO: Add your comment here *)
FUNCTION CanPlayerCapture

//	CanPlayerCapture := FALSE;

//	FOR Row := 1 TO 8 DO
//
	//	FOR Column := 1 TO 8 DO

		//	Piece := Board[Row, Column];

			//CASE PlayerColor OF

			//	WHITE_COLOR:

			//		IF (Piece = WHITE) OR
			//			(Piece = WHITE_KING) THEN

			////			IF CheckRegularCapture(
			//				FromRow := Row,
			//				FromColumn := Column,
			//				ToRow := Row + 2,
			//				ToColumn := Column + 2,
			//				Piece := Piece,
			//				Board := Board) THEN
//
			//				CanPlayerCapture := TRUE;
			//				RETURN;

			//			END_IF;

			//			IF CheckRegularCapture(
			//				FromRow := Row,
			//				FromColumn := Column,
			//				ToRow := Row + 2,
			//				ToColumn := Column - 2,
			//				Piece := Piece,
			//				Board := Board) THEN

			//				CanPlayerCapture := TRUE;
			//				RETURN;

			//			END_IF;

			//			IF Piece = WHITE_KING THEN

			//				IF CheckRegularCapture(
			//					FromRow := Row,
			//					FromColumn := Column,
			//					ToRow := Row - 2,
			//					ToColumn := Column + 2,
			//					Piece := Piece,
			//					Board := Board) THEN

			//					CanPlayerCapture := TRUE;
			//					RETURN;

			//				END_IF;

			//				IF CheckRegularCapture(
			//					FromRow := Row,
			//					FromColumn := Column,
			///					ToRow := Row - 2,
			//					ToColumn := Column - 2,
			//					Piece := Piece,
			//					Board := Board) THEN

			//					CanPlayerCapture := TRUE;
			//					RETURN;

			//				END_IF;

			//			END_IF;
//
			//		END_IF;

			//	BLACK_COLOR:

			//		IF (Piece = BLACK) OR
			//			(Piece = BLACK_KING) THEN
//
			//			IF CheckRegularCapture(
			//				FromRow := Row,
			///				FromColumn := Column,
			//				ToRow := Row - 2,
			//				ToColumn := Column + 2,
			//				Piece := Piece,
			//				Board := Board) THEN
//
//							CanPlayerCapture := TRUE;
//							RETURN;
//
//						END_IF;
//
//						IF CheckRegularCapture(
//							FromRow := Row,
//							FromColumn := Column,
//							ToRow := Row - 2,
//							ToColumn := Column - 2,
//							Piece := Piece,
//							Board := Board) THEN

//							CanPlayerCapture := TRUE;
//							RETURN;

//						END_IF;

//						IF Piece = BLACK_KING THEN
//
//							IF CheckRegularCapture(
//								FromRow := Row,
//								FromColumn := Column,
//								ToRow := Row + 2,
///								ToColumn := Column + 2,
//								Piece := Piece,
//								Board := Board) THEN
//
//								CanPlayerCapture := TRUE;
//								RETURN;
//
//							END_IF;

//							IF CheckRegularCapture(
//								FromRow := Row,
//								FromColumn := Column,
//								ToRow := Row + 2,
//								ToColumn := Column - 2,
//								Piece := Piece,
//								Board := Board) THEN
//
//								CanPlayerCapture := TRUE;
//								RETURN;
//
//							END_IF;
//
//						END_IF;
//
//					END_IF;
//
//			END_CASE;

//		END_FOR;

//	END_FOR;

END_FUNCTION
```

#### FB_InitGame.st
```iecst
(* TODO: Add your comment here *)
FUNCTION_BLOCK FB_InitGame
	IF Execute THEN

		MovesWithoutCapture := 0;
		PlayerColor := WHITE_COLOR;
		Winner := NONE;
		GameState := CHECKING_BOARD;

		Done := TRUE;

	ELSE
		Done := FALSE;
	END_IF;
END_FUNCTION_BLOCK
```

#### FB_InitBoard.st
```iecst
(* TODO: Add your comment here *)
FUNCTION_BLOCK FB_InitBoard
	IF Execute THEN

		(* Wyczyszczenie planszy *)
		FOR Row := 1 TO 8 DO
			FOR Column := 1 TO 8 DO
				BoardBoard[Row, Column] := EMPTY;
			END_FOR;
		END_FOR;

		(* Ustawienie białych pionków *)
		FOR Column := 1 TO 8 DO

			IF (Column MOD 2) = 1 THEN
				BoardBoard[1, Column] := WHITE;
				BoardBoard[3, Column] := WHITE;
			ELSE
				BoardBoard[2, Column] := WHITE;
			END_IF;

		END_FOR;

		(* Ustawienie czarnych pionków *)
		FOR Column := 1 TO 8 DO

			IF (Column MOD 2) = 0 THEN
				BoardBoard[6, Column] := BLACK;
				BoardBoard[8, Column] := BLACK;
			ELSE
				BoardBoard[7, Column] := BLACK;
			END_IF;

		END_FOR;

		GameState := WAITING_PLAYER;

		Done := TRUE;

	ELSE

		Done := FALSE;

	END_IF;
END_FUNCTION_BLOCK
```

#### CanPieceCaptureAgain.st
```iecst
(* TODO: Add your comment here *)
FUNCTION CanPieceCaptureAgain
	CanPieceCaptureAgain := FALSE;

	CASE Piece OF

		WHITE:

			IF CheckRegularCapture(
				FromRow := Row,
				FromColumn := Column,
				ToRow := Row + 2,
				ToColumn := Column + 2,
				Piece := Piece,
				Board := Board) THEN

				CanPieceCaptureAgain := TRUE;
				RETURN;

			END_IF;

			IF CheckRegularCapture(
				FromRow := Row,
				FromColumn := Column,
				ToRow := Row + 2,
				ToColumn := Column - 2,
				Piece := Piece,
				Board := Board) THEN

				CanPieceCaptureAgain := TRUE;
				RETURN;

			END_IF;

		BLACK:

			IF CheckRegularCapture(
				FromRow := Row,
				FromColumn := Column,
				ToRow := Row - 2,
				ToColumn := Column + 2,
				Piece := Piece,
				Board := Board) THEN

				CanPieceCaptureAgain := TRUE;
				RETURN;

			END_IF;

			IF CheckRegularCapture(
				FromRow := Row,
				FromColumn := Column,
				ToRow := Row - 2,
				ToColumn := Column - 2,
				Piece := Piece,
				Board := Board) THEN

				CanPieceCaptureAgain := TRUE;
				RETURN;

			END_IF;

			WHITE_KING,
		BLACK_KING:

			IF CheckRegularCapture(
				FromRow := Row,
				FromColumn := Column,
				ToRow := Row + 2,
				ToColumn := Column + 2,
				Piece := Piece,
				Board := Board) THEN

				CanPieceCaptureAgain := TRUE;
				RETURN;

			END_IF;

			IF CheckRegularCapture(
				FromRow := Row,
				FromColumn := Column,
				ToRow := Row + 2,
				ToColumn := Column - 2,
				Piece := Piece,
				Board := Board) THEN

				CanPieceCaptureAgain := TRUE;
				RETURN;

			END_IF;

			IF CheckRegularCapture(
				FromRow := Row,
				FromColumn := Column,
				ToRow := Row - 2,
				ToColumn := Column + 2,
				Piece := Piece,
				Board := Board) THEN

				CanPieceCaptureAgain := TRUE;
				RETURN;

			END_IF;

			IF CheckRegularCapture(
				FromRow := Row,
				FromColumn := Column,
				ToRow := Row - 2,
				ToColumn := Column - 2,
				Piece := Piece,
				Board := Board) THEN

				CanPieceCaptureAgain := TRUE;
				RETURN;

			END_IF;

	END_CASE;
END_FUNCTION
```

#### FB_PromotePiece.st
```iecst
(* TODO: Add your comment here *)
FUNCTION_BLOCK FB_PromotePiece

	IF Execute THEN

		CASE Board[Row, Column] OF

			WHITE:

				IF Row = 8 THEN
					Board[Row, Column] := WHITE_KING;
				END_IF;

			BLACK:

				IF Row = 1 THEN
					Board[Row, Column] := BLACK_KING;
				END_IF;

		END_CASE;

		Done := TRUE;

	ELSE

		Done := FALSE;

	END_IF;

END_FUNCTION_BLOCK
```

### Program Logical/Programs/Robot-programy

#### move.st
```iecst
VAR {AT 'MotionCtrl'}
    StartPoint {ACCESS 'STMotionStartPoint'}: McPointType;
    EndPoint {ACCESS 'STMotionEndPoint'}: McPointType;
    HomePoint {ACCESS 'STMotionHomePoint'}: McPointType;
    Done {ACCESS 'STMotionDone'}: BOOL;
END_VAR

//VAR {AT PLC}
//    doMagnet : BOOL;
//    MagnetStatus : BOOL;
//END_VAR

VAR
    Offs : McPosType := (Z:=20);

    StartPointOffs : McPointType;
    EndPointOffs : McPointType;
END_VAR

PROGRAM _MAIN
    Done := FALSE;
    Feedrate(5000);

    StartPointOffs := StartPoint;
    StartPointOffs.Pos.Z := StartPointOffs.Pos.Z + Offs.Z;
    EndPointOffs := EndPoint;
    EndPointOffs.Pos.Z := EndPointOffs.Pos.Z + Offs.Z;

    MoveJ(StartPointOffs);
    MoveL(StartPoint);
    WaitEndMove();
    //doMagnet := TRUE;
    //WaitUntil(MagnetStatus);
    MoveL(StartPointOffs); // zapytac sie czy tutaj da sie dac StartPoint + Offs, dla krotszego kodu

    MoveJ(HomePoint);

    MoveJ(EndPointOffs);
    MoveL(EndPoint);
    WaitEndMove();
    //doMagnet := FALSE;
    //WaitUntil(NOT MagnetStatus);
    MoveL(EndPointOffs);

    MoveJ(HomePoint);

    WaitEndMove();
    Done := TRUE;
END_PROGRAM
```

### Program Logical/Programs/TestOpcua

#### Variables.var
```iecst
VAR
	j : USINT;
	i : USINT;
END_VAR
```

#### Main.st
```iecst
PROGRAM _INIT
	gTrudnosc := 0;
	gBoard[0,1] := 2;
	gBoard[0,3] := 2;
	gBoard[0,5] := 2;
	gBoard[0,7] := 2;

	gBoard[1,0] := 2;
	gBoard[1,2] := 2;
	gBoard[1,4] := 2;
	gBoard[1,6] := 2;

	gBoard[2,1] := 2;
	gBoard[2,3] := 2;
	gBoard[2,5] := 2;
	gBoard[2,7] := 2;

	gBoard[5,0] := 1;
	gBoard[5,2] := 1;
	gBoard[5,4] := 1;
	gBoard[5,6] := 1;

	gBoard[6,1] := 1;
	gBoard[6,3] := 1;
	gBoard[6,5] := 1;
	gBoard[6,7] := 1;

	gBoard[7,0] := 1;
	gBoard[7,2] := 1;
	gBoard[7,4] := 1;
	gBoard[7,6] := 1;
	gGraStart := FALSE;
	gJakiKolor := FALSE;

END_PROGRAM

PROGRAM _CYCLIC
	(* Insert code here *)
	gTest;
END_PROGRAM

PROGRAM _EXIT
	(* Insert code here *)

END_PROGRAM
```

Listed in the project but not available here: Logical/Libraries/CameraMath/Types.typ, Logical/Libraries/CameraMath/Constants.var, Logical/Programs/Motion/RobotMovements/Types.typ, Logical/Programs/Alarms, Logical/Programs/CheckLegal/Types.typ, Logical/Programs/CheckLegal/CanPlayerCapture.st, Logical/Programs/PieceMovementProgram/Types.typ, Logical/Programs/PieceMovementProgram/CheckRegularCapture.st
